# EPICS substitutions: iocBoot/ioc13ida/auto_shutter.substitutions
file "$(CARS)/CARSApp/Db/auto_shutter.db"
{
pattern
{P,      SHUT, SHUT_STATUS,       SHUT_CONTROL,        PERIOD, BEAM_READY}
{13IDA:, FOE,  13IDA:eps_mbbi25,  13IDA:OpenFEShutter, 30,    PA:13ID:STA_A_BEAMREADY_PL}
{13IDA:, IDCD, 13IDA:eps_mbbi26,  13IDA:OpenCDShutter, 30,    PA:13ID:STA_C_BEAMREADY_PL}
{13IDA:, IDE,  13IDA:eps_mbbi27,  13IDA:OpenEShutter,  30,    PA:13ID:STA_E_BEAMREADY_PL}
}
